(****************************************************************************************)
(*							Beckhoff Automation Poland									*)
(*							L_TBConvArrBitsToDword  v1.0								*)
(*									7.04.2009											*)
(*		This function converts array 32 single bits into a value of type ”double word”	*)
(*______________________________________________________________________________________*)
FUNCTION L_TBConvArrBitsToDword : DWORD
VAR_INPUT
	arrBits: ARRAY [0..31] OF BOOL;
END_VAR

L_TBConvArrBitsToDword.0 := arrBits[0];
L_TBConvArrBitsToDword.1 := arrBits[1];
L_TBConvArrBitsToDword.2 := arrBits[2];
L_TBConvArrBitsToDword.3 := arrBits[3];
L_TBConvArrBitsToDword.4 := arrBits[4];
L_TBConvArrBitsToDword.5 := arrBits[5];
L_TBConvArrBitsToDword.6 := arrBits[6];
L_TBConvArrBitsToDword.7 := arrBits[7];
L_TBConvArrBitsToDword.8 := arrBits[8];
L_TBConvArrBitsToDword.9 := arrBits[9];
L_TBConvArrBitsToDword.10 := arrBits[10];
L_TBConvArrBitsToDword.11 := arrBits[11];
L_TBConvArrBitsToDword.12 := arrBits[12];
L_TBConvArrBitsToDword.13 := arrBits[13];
L_TBConvArrBitsToDword.14 := arrBits[14];
L_TBConvArrBitsToDword.15 := arrBits[15];
L_TBConvArrBitsToDword.16 := arrBits[16];
L_TBConvArrBitsToDword.17 := arrBits[17];
L_TBConvArrBitsToDword.18 := arrBits[18];
L_TBConvArrBitsToDword.19 := arrBits[19];
L_TBConvArrBitsToDword.20 := arrBits[20];
L_TBConvArrBitsToDword.21 := arrBits[21];
L_TBConvArrBitsToDword.22 := arrBits[22];
L_TBConvArrBitsToDword.23 := arrBits[23];
L_TBConvArrBitsToDword.24 := arrBits[24];
L_TBConvArrBitsToDword.25 := arrBits[25];
L_TBConvArrBitsToDword.26 := arrBits[26];
L_TBConvArrBitsToDword.27 := arrBits[27];
L_TBConvArrBitsToDword.28 := arrBits[28];
L_TBConvArrBitsToDword.29 := arrBits[29];
L_TBConvArrBitsToDword.30 := arrBits[30];
L_TBConvArrBitsToDword.31 := arrBits[31];

END_FUNCTION

(* stored: Version 1.1.0.1, ProductVersion 3.1.4026.13, FileIdentifier f506ec5fff6630a7d4ebebeddc0e281a58dd122e, FileSignature 39ec7a94515886e5603dbd87ff9bbfc3f34075567353c1ee0ab2f08ac423efc0b081336024b82fcebae77f106a9befe405e99c915b386d3e65aa8b63b8b29a2c81a3ca877fa7e801b206e24125c309cdba29e80a256f3b77b9fe13fce902f33756413875fc2a3f260055f6f7fc07bf22306992ae27c5096405db681d8ebc0285aad60d9da33cc2223583b647614bac53560806b8ea7ef659abfac62ade9eb1780385a31b493491a2ef2cb4472b574876e7f7521c6e8f3de025275e17a050a55d3b73fefd116fb77c226e0f6ae7755f9199d0c6f268206890f5fdcd065c88cef06dbdfffac098d2e2259c1e52f3086b3cb4e8f6a7ccc4a6cb70ca0c277ff2cf4f
   POU L_TBConvArrBitsToDword: Id {b131d12c-c182-43ce-83b0-735883441a42}, SpecialFunc None *)
